PROGRAM MAIN
VAR
	//nState: UINT := 0;
	Axis : ARRAY [0..3] OF ARRAY [0..1] OF AXIS_REF;
	MoveAbsolute : MC_MoveAbsolute;
	MoveRelative : MC_MoveRelative;
	MoveHome : MC_Home;
	WriteParameter : MC_WriteParameter;
	ReadParameter : MC_ReadParameter;
	AxisPower : MC_Power;
	Reset : MC_Reset;
	FB_Functions : FB_Functions;
	AxisParams : MC_AxisParameter;
	ReadDriveAddress : MC_ReadDriveAddress;
	SetControlLoop : MC_SelectControlLoop;
	ReadBoolParameter : MC_ReadBoolParameter;
	WriteBoolParameter : MC_WriteBoolParameter;
	SetActualPosition : MC_SetPosition;
	Axis1LoopID : UINT;
	Axis2LoopID : UINT;
	Axis3LoopID : UINT;
	Axis4LoopID : UINT;
	activeAxisLoopID : ARRAY [0..3] OF UINT;
END_VAR

//Axis1[0]();
//Axis1[1]();
//Axis1[2]();
//Axis1();

Axis[0][0](); // incremental encoder axis 1
Axis[0][1](); // absolute encoder axis 1
activeAxisLoopID[0] := Axis[0][0].NcToPlc.ActiveControlLoopIndex;

Axis[1][0](); // incremental encoder axis 2
Axis[1][1](); // absolute encoder axis 2
activeAxisLoopID[1] := Axis[1][0].NcToPlc.ActiveControlLoopIndex;

Axis[2][0](); // incremental encoder axis 3
Axis[2][1](); // absolute encoder axis 3
activeAxisLoopID[2] := Axis[2][0].NcToPlc.ActiveControlLoopIndex;

Axis[3][0](); // incremental encoder axis 4
Axis[3][1](); // absolute encoder axis 4
activeAxisLoopID[3] := Axis[3][0].NcToPlc.ActiveControlLoopIndex;



//E_NcEncoderType.NcEncoderType_Simulation

//CASE nState OF
//	0:
//	nState := 10;
//	
//	10:
//	MoveAbsolute(Axis:=Axis1[0],Execute:=FALSE);
//	Reset(Axis:=Axis1[0],Execute:=FALSE);
//	nState := 20;
//	
//	20:
//	AxisPower(Axis:=Axis1[0],
//			Enable:=TRUE,
//			Enable_Positive:=TRUE,
//			Enable_Negative:=TRUE);
//			
//	IF GVL_VARS1.execute THEN
//		nState := 30;
//	END_IF
//
//	
//	30:
//	MoveAbsolute(Axis:=Axis1[0],
//					Position:=GVL_VARS1.position,
//					Velocity:=GVL_VARS1.velocity);
//	MoveAbsolute(Axis:=Axis1[0],
//					Execute:=TRUE);		
//	IF MoveAbsolute.Done THEN
//		MoveAbsolute(Axis:=Axis1[0],Execute:=FALSE);
//	END_IF
//	GVL_VARS1.execute := FALSE;
//	nState := 10;
//END_CASE


//AxisPower(Axis:=Axis1);
//MoveAbsolute(Axis:=Axis1);
//Reset(Axis:=Axis1);

END_PROGRAM

(* stored: Version 1.1.0.1, ProductVersion 3.1.4024.12
   POU MAIN: Id {f070e0eb-d52d-4666-8d92-3578df9d3e28}, SpecialFunc None *)
